FUNCTION_BLOCK FB_InstrumentDetect
VAR_INPUT
END_VAR
VAR_OUTPUT
END_VAR
VAR
	m_instruOnCounts :INT :=0;
	m_InstruOnCountThres :INT :=50;
END_VAR

// check if instrument is on
METHOD run : BOOL
VAR_INPUT
	IOValue :UDINT;
END_VAR
//Instrument single   At installation--2#0*0*   not installation --2#1*1*  And Hall single --2#100 0000
IF (IOValue AND 16#4A) = 64 OR (IOValue AND 16#4A) = 0  THEN
	m_instruOnCounts := MIN( m_instruOnCounts +1,m_InstruOnCountThres);
ELSIF (IOValue AND 16#4A) = 10  THEN
	m_instruOnCounts :=0;
END_IF
run := m_instruOnCounts >= m_InstruOnCountThres;
END_METHOD

END_FUNCTION_BLOCK

(* stored: Version 1.1.0.1, ProductVersion 3.1.4024.11
   POU FB_InstrumentDetect: Id {b69ad326-ec41-4095-b403-6a4f502c7c86}, SpecialFunc None
   Method run: Id {2a4a25fd-8c3e-4d43-b812-7646c7f18efc} *)
